(* IEC 61131-3 sources: RL_MAR/experiments/comparison/llm4plc/results/gpt-4o-mini_20260506_100619/20260506_102345, 4 files *)

(* ---- generated_code_iteration_0.st ---- *)
ructured-text
START_ST
FUNCTION_BLOCK WindowCleaningSystem
VAR_INPUT
    StartButton : BOOL;
    EmergencyStop : BOOL;
    UpperLimit : BOOL;
    LowerLimit : BOOL;
END_VAR

VAR_OUTPUT
    ElevatorUp : BOOL;
    ElevatorDown : BOOL;
    RotateClockwise : BOOL;
    WaterPump : BOOL;
END_VAR

VAR
    state : INT; // THE STATE VARIABLE
    CleaningInProgress : BOOL; // FLAG TO INDICATE IF CLEANING IS IN PROGRESS
END_VAR

// STATE DECLARATIONS
CONSTANT
    STATE_IDLE : INT := 0;
    STATE_MOVING_UP : INT := 1;
    STATE_CLEANING : INT := 2;
    STATE_MOVING_DOWN : INT := 3;
    STATE_EMERGENCY_STOP : INT := 4;
END_CONSTANT

// INITIALIZE THE FUNCTION BLOCK
state := STATE_IDLE;
CleaningInProgress := FALSE;

// IMPLEMENT THE STATE MACHINE LOGIC
CASE state OF
    STATE_IDLE:
        ElevatorUp := FALSE;
        ElevatorDown := FALSE;
        RotateClockwise := FALSE;
        WaterPump := FALSE;

        IF StartButton = TRUE AND EmergencyStop = FALSE AND CleaningInProgress = FALSE THEN
            state := STATE_MOVING_UP;
        END_IF;

    STATE_MOVING_UP:
        ElevatorUp := TRUE;
        ElevatorDown := FALSE;
        RotateClockwise := FALSE;
        WaterPump := FALSE;

        IF UpperLimit = TRUE THEN
            state := STATE_CLEANING;
            CleaningInProgress := TRUE;
        END_IF;

        IF EmergencyStop = TRUE THEN
            state := STATE_EMERGENCY_STOP;
        END_IF;

    STATE_CLEANING:
        ElevatorUp := FALSE;
        ElevatorDown := FALSE;
        RotateClockwise := TRUE;
        WaterPump := TRUE;

        IF LowerLimit = TRUE THEN
            state := STATE_MOVING_DOWN;
        END_IF;

        IF EmergencyStop = TRUE THEN
            state := STATE_EMERGENCY_STOP;
        END_IF;

    STATE_MOVING_DOWN:
        ElevatorUp := FALSE;
        ElevatorDown := TRUE;
        RotateClockwise := FALSE;
        WaterPump := FALSE;

        IF LowerLimit = TRUE AND CleaningInProgress = TRUE THEN
            state := STATE_IDLE;
            CleaningInProgress := FALSE;
        END_IF;

        IF EmergencyStop = TRUE THEN
            state := STATE_EMERGENCY_STOP;
        END_IF;

    STATE_EMERGENCY_STOP:
        ElevatorUp := FALSE;
        ElevatorDown := FALSE;
        RotateClockwise := FALSE;
        WaterPump := FALSE;

        // Stay in emergency stop state until reset
        IF EmergencyStop = FALSE THEN
            state := STATE_IDLE; // Reset to idle state when emergency stop is released
        END_IF;

END_CASE;

END_FUNCTION_BLOCK
END_ST

(* ---- generated_code_iteration_1.st ---- *)
START_REASON
The errors in the original Structured Text (ST) code occurred because the variable section was incorrectly defined with "VAR_OUTPUT" and "VAR_INPUT" instead of just "VAR". In addition, the use of "CONSTANT" was not valid in the context it was placed. The correct approach is to define constants within the variable section. This ensures proper syntax and structure according to the requirements of the Structured Text language.
END_REASON

START_ST
FUNCTION_BLOCK WindowCleaningSystem
VAR_INPUT
    StartButton : BOOL;
    EmergencyStop : BOOL;
    UpperLimit : BOOL;
    LowerLimit : BOOL;
END_VAR

VAR_OUTPUT
    ElevatorUp : BOOL;
    ElevatorDown : BOOL;
    RotateClockwise : BOOL;
    WaterPump : BOOL;
END_VAR

VAR
    state : INT; // THE STATE VARIABLE
    CleaningInProgress : BOOL; // FLAG TO INDICATE IF CLEANING IS IN PROGRESS

    // STATE DECLARATIONS
    STATE_IDLE : INT := 0;
    STATE_MOVING_UP : INT := 1;
    STATE_CLEANING : INT := 2;
    STATE_MOVING_DOWN : INT := 3;
    STATE_EMERGENCY_STOP : INT := 4;
END_VAR

// INITIALIZE THE FUNCTION BLOCK
state := STATE_IDLE;
CleaningInProgress := FALSE;

// IMPLEMENT THE STATE MACHINE LOGIC
CASE state OF
    STATE_IDLE:
        ElevatorUp := FALSE;
        ElevatorDown := FALSE;
        RotateClockwise := FALSE;
        WaterPump := FALSE;

        IF StartButton = TRUE AND EmergencyStop = FALSE AND CleaningInProgress = FALSE THEN
            state := STATE_MOVING_UP;
        END_IF;

    STATE_MOVING_UP:
        ElevatorUp := TRUE;
        ElevatorDown := FALSE;
        RotateClockwise := FALSE;
        WaterPump := FALSE;

        IF UpperLimit = TRUE THEN
            state := STATE_CLEANING;
            CleaningInProgress := TRUE;
        END_IF;

        IF EmergencyStop = TRUE THEN
            state := STATE_EMERGENCY_STOP;
        END_IF;

    STATE_CLEANING:
        ElevatorUp := FALSE;
        ElevatorDown := FALSE;
        RotateClockwise := TRUE;
        WaterPump := TRUE;

        IF LowerLimit = TRUE THEN
            state := STATE_MOVING_DOWN;
        END_IF;

        IF EmergencyStop = TRUE THEN
            state := STATE_EMERGENCY_STOP;
        END_IF;

    STATE_MOVING_DOWN:
        ElevatorUp := FALSE;
        ElevatorDown := TRUE;
        RotateClockwise := FALSE;
        WaterPump := FALSE;

        IF LowerLimit = TRUE AND CleaningInProgress = TRUE THEN
            state := STATE_IDLE;
            CleaningInProgress := FALSE;
        END_IF;

        IF EmergencyStop = TRUE THEN
            state := STATE_EMERGENCY_STOP;
        END_IF;

    STATE_EMERGENCY_STOP:
        ElevatorUp := FALSE;
        ElevatorDown := FALSE;
        RotateClockwise := FALSE;
        WaterPump := FALSE;

        // Stay in emergency stop state until reset
        IF EmergencyStop = FALSE THEN
            state := STATE_IDLE; // Reset to idle state when emergency stop is released
        END_IF;

END_CASE;

END_FUNCTION_BLOCK
END_ST

(* ---- generated_code_iteration_2.st ---- *)
START_REASON
The errors in the original Structured Text (ST) code occurred primarily due to the incorrect use of variable sections. The sections labeled as "VAR_INPUT" and "VAR_OUTPUT" should be simply labeled as "VAR" to conform to the requirements. Additionally, the error message indicated that the CASE statement requires constant integer values, which means that the state variables should be defined as constants within the variable section. This ensures that the CASE statement can properly reference these states.
END_REASON

START_ST
FUNCTION_BLOCK WindowCleaningSystem
VAR
    StartButton : BOOL;
    EmergencyStop : BOOL;
    UpperLimit : BOOL;
    LowerLimit : BOOL;

    ElevatorUp : BOOL;
    ElevatorDown : BOOL;
    RotateClockwise : BOOL;
    WaterPump : BOOL;

    state : INT; // THE STATE VARIABLE
    CleaningInProgress : BOOL; // FLAG TO INDICATE IF CLEANING IS IN PROGRESS

    // STATE DECLARATIONS
    STATE_IDLE : INT := 0;
    STATE_MOVING_UP : INT := 1;
    STATE_CLEANING : INT := 2;
    STATE_MOVING_DOWN : INT := 3;
    STATE_EMERGENCY_STOP : INT := 4;
END_VAR

// INITIALIZE THE FUNCTION BLOCK
state := STATE_IDLE;
CleaningInProgress := FALSE;

// IMPLEMENT THE STATE MACHINE LOGIC
CASE state OF
    STATE_IDLE:
        ElevatorUp := FALSE;
        ElevatorDown := FALSE;
        RotateClockwise := FALSE;
        WaterPump := FALSE;

        IF StartButton = TRUE AND EmergencyStop = FALSE AND CleaningInProgress = FALSE THEN
            state := STATE_MOVING_UP;
        END_IF;

    STATE_MOVING_UP:
        ElevatorUp := TRUE;
        ElevatorDown := FALSE;
        RotateClockwise := FALSE;
        WaterPump := FALSE;

        IF UpperLimit = TRUE THEN
            state := STATE_CLEANING;
            CleaningInProgress := TRUE;
        END_IF;

        IF EmergencyStop = TRUE THEN
            state := STATE_EMERGENCY_STOP;
        END_IF;

    STATE_CLEANING:
        ElevatorUp := FALSE;
        ElevatorDown := FALSE;
        RotateClockwise := TRUE;
        WaterPump := TRUE;

        IF LowerLimit = TRUE THEN
            state := STATE_MOVING_DOWN;
        END_IF;

        IF EmergencyStop = TRUE THEN
            state := STATE_EMERGENCY_STOP;
        END_IF;

    STATE_MOVING_DOWN:
        ElevatorUp := FALSE;
        ElevatorDown := TRUE;
        RotateClockwise := FALSE;
        WaterPump := FALSE;

        IF LowerLimit = TRUE AND CleaningInProgress = TRUE THEN
            state := STATE_IDLE;
            CleaningInProgress := FALSE;
        END_IF;

        IF EmergencyStop = TRUE THEN
            state := STATE_EMERGENCY_STOP;
        END_IF;

    STATE_EMERGENCY_STOP:
        ElevatorUp := FALSE;
        ElevatorDown := FALSE;
        RotateClockwise := FALSE;
        WaterPump := FALSE;

        // Stay in emergency stop state until reset
        IF EmergencyStop = FALSE THEN
            state := STATE_IDLE; // Reset to idle state when emergency stop is released
        END_IF;

END_CASE;

END_FUNCTION_BLOCK
END_ST

(* ---- generated_code_iteration_3.st ---- *)
START_REASON
The errors in the original Structured Text (ST) code occurred due to the incorrect use of variable sections and the requirement for the CASE statement to reference constant integer values. The variable section should be labeled simply as "VAR" instead of using specific input or output labels. Additionally, the state variables used in the CASE statement must be defined as constants to ensure compliance with the requirements of the CASE statement. This ensures that the CASE statement can properly reference these states without causing compilation errors.
END_REASON

START_ST
FUNCTION_BLOCK WindowCleaningSystem
VAR
    StartButton : BOOL;
    EmergencyStop : BOOL;
    UpperLimit : BOOL;
    LowerLimit : BOOL;

    ElevatorUp : BOOL;
    ElevatorDown : BOOL;
    RotateClockwise : BOOL;
    WaterPump : BOOL;

    state : INT; // THE STATE VARIABLE
    CleaningInProgress : BOOL; // FLAG TO INDICATE IF CLEANING IS IN PROGRESS
END_VAR

// STATE DECLARATIONS
CONST
    STATE_IDLE : INT := 0;
    STATE_MOVING_UP : INT := 1;
    STATE_CLEANING : INT := 2;
    STATE_MOVING_DOWN : INT := 3;
    STATE_EMERGENCY_STOP : INT := 4;
END_CONST

// INITIALIZE THE FUNCTION BLOCK
state := STATE_IDLE;
CleaningInProgress := FALSE;

// IMPLEMENT THE STATE MACHINE LOGIC
CASE state OF
    STATE_IDLE:
        ElevatorUp := FALSE;
        ElevatorDown := FALSE;
        RotateClockwise := FALSE;
        WaterPump := FALSE;

        IF StartButton = TRUE AND EmergencyStop = FALSE AND CleaningInProgress = FALSE THEN
            state := STATE_MOVING_UP;
        END_IF;

    STATE_MOVING_UP:
        ElevatorUp := TRUE;
        ElevatorDown := FALSE;
        RotateClockwise := FALSE;
        WaterPump := FALSE;

        IF UpperLimit = TRUE THEN
            state := STATE_CLEANING;
            CleaningInProgress := TRUE;
        END_IF;

        IF EmergencyStop = TRUE THEN
            state := STATE_EMERGENCY_STOP;
        END_IF;

    STATE_CLEANING:
        ElevatorUp := FALSE;
        ElevatorDown := FALSE;
        RotateClockwise := TRUE;
        WaterPump := TRUE;

        IF LowerLimit = TRUE THEN
            state := STATE_MOVING_DOWN;
        END_IF;

        IF EmergencyStop = TRUE THEN
            state := STATE_EMERGENCY_STOP;
        END_IF;

    STATE_MOVING_DOWN:
        ElevatorUp := FALSE;
        ElevatorDown := TRUE;
        RotateClockwise := FALSE;
        WaterPump := FALSE;

        IF LowerLimit = TRUE AND CleaningInProgress = TRUE THEN
            state := STATE_IDLE;
            CleaningInProgress := FALSE;
        END_IF;

        IF EmergencyStop = TRUE THEN
            state := STATE_EMERGENCY_STOP;
        END_IF;

    STATE_EMERGENCY_STOP:
        ElevatorUp := FALSE;
        ElevatorDown := FALSE;
        RotateClockwise := FALSE;
        WaterPump := FALSE;

        // Stay in emergency stop state until reset
        IF EmergencyStop = FALSE THEN
            state := STATE_IDLE; // Reset to idle state when emergency stop is released
        END_IF;

END_CASE;

END_FUNCTION_BLOCK
END_ST
